{attribute 'GeneratedUsingTerminal: EL5072-0000-0016'}
{attribute addProperty BoxType "EL5072-0000-0016"}
{attribute addProperty Description "EL5072 2Ch. Inductive sensor interface (LVDT, Half Bridge)"}
{attribute addProperty Physics "KK"}
{attribute addProperty Id "IND_Inputs_Channel_1AT %I*IND_Inputs_Channel_BBE8401F18IND_Inputs_Channel_2AT %I*IND_Inputs_Channel_BBE8401F18IND_Outputs_Channel_1AT %Q*IND_Outputs_Channel_02FDE6C97IND_Outputs_Channel_2AT %Q*IND_Outputs_Channel_02FDE6C97WcStateAT %I*WcState_9091E0EB2InfoDataAT %I*InfoData_32EB74EA10"}
{attribute addProperty CRC "410576726"}
{attribute addProperty Size "62"}
TYPE EL5072_1878E756 EXTENDS EtcSlaveTerminalBase_947E5A46 :
STRUCT
	{attribute addProperty Name "IND_Inputs_Channel_1"}
	IND_Inputs_Channel_1 : IND_Inputs_Channel_BBE8401F;
	{attribute addProperty Name "IND_Inputs_Channel_2"}
	IND_Inputs_Channel_2 : IND_Inputs_Channel_BBE8401F;
	{attribute addProperty Name "IND_Outputs_Channel_1"}
	IND_Outputs_Channel_1 : IND_Outputs_Channel_02FDE6C9;
	{attribute addProperty Name "IND_Outputs_Channel_2"}
	IND_Outputs_Channel_2 : IND_Outputs_Channel_02FDE6C9;
	{attribute addProperty Name "WcState"}
	WcState : WcState_9091E0EB;
	{attribute addProperty Name "InfoData"}
	InfoData : InfoData_32EB74EA;
END_STRUCT
END_TYPE

(* stored: Version 1.2.0.0, ProductVersion 3.1.4024.11
   DUT EL5072_1878E756: Id {aa122d2c-043b-473a-a354-375bae6edd42} *)
